(* CODESYS project WagoLibAwsIotThingShadow_v0.0.1.library
   Company: WAGO Corp. USA
   Title: WagoLibAwsIotThingShadow
   Description: This library contains function blocks which allow the project to interact directly with AWS IoT Thing Shadow document.
   Author: Jesse Cox
   Version: 0.0.1

Project tree, tasks and I/O mapping:
  libraries: SysProcess, 3.5.7.0 (System); WagoSysString, 1.6.0.0 (WAGO); WagoAppFileDir, * (WAGO); SysTypes2 Interfaces, 3.5.4.0 (System)
  text list GlobalTextList
  data type typIOT_THING_SHADOW
  function block GET_AWS_IOT_THING_SHADOW [ST]: CURL_STRING
  function block UPDATE_AWS_IOT_THING_SHADOW [ST]: PUB_STRING
*)

// typIOT_THING_SHADOW
TYPE typIOT_THING_SHADOW :
STRUCT
		sLabel	: STRING;
		sValue	: STRING;
END_STRUCT
END_TYPE

// GET_AWS_IOT_THING_SHADOW
FUNCTION_BLOCK GET_AWS_IOT_THING_SHADOW	
VAR_IN_OUT
	xExecute: BOOL;
	Shadow_Attributes	: ARRAY[*] OF typIOT_THING_SHADOW;
END_VAR
VAR_INPUT
	sThingName			: STRING;
	sRootCaPath			: STRING;
	sCertPath			: STRING;
	sKeyPath			: STRING;
	sEndpoint			: STRING;
END_VAR
VAR_OUTPUT
	//diTest				: DINT;
END_VAR
VAR
	sQueryBashScript	: STRING(255);
	sBashResponse: STRING;
	ptBashRslt: RTS_IEC_RESULT;
	diFileStatus: DINT;
	fbReadShadowFile: FbReadWholeFile_cpt;
	oReadFileStatus: FbResult;
	xReadFileTrig: BOOL;
	xREadFileError: BOOL;
	xREadFileBusy: BOOL;
	abFileData		: ARRAY[1..10000] OF BYTE;
	udiReadFileSize: UDINT := 10000;
	udiReadRxNumOfBytes: UDINT;
	xReadFileEndReached: BOOL;
	xConvertToTyp: BOOL;
	b: UDINT;
	xByteIsChar: BOOL;
	iCurlIndex: INT;
	xOnLabel: BOOL;
	xOnValue: BOOL;
	iWriteIndex: INT;
	sCurrentValueString: STRING;
	sCurrentLabelString: STRING;
	ub: DINT;
END_VAR

ub:=UPPER_BOUND (Shadow_Attributes,1);

IF xExecute THEN
	sQueryBashScript := CURL_STRING(
							sThingName:= sThingName, 
							sRootCaPath:= sRootCaPath, 
							sCertPath:= sCertPath, 
							sKeyPath:= sKeyPath, 
							sEndPoint:= sEndpoint);
	diFileStatus := SysProcessExecuteCommand2(pszCommand:= sQueryBashScript, pszStdOut:= sBashResponse, udiStdOutLen:= 255, pResult:= ptBashRslt);
	
	//diTest := diFileStatus;
	IF (diFileStatus <> 0) AND NOT xReadFileEndReached THEN
		xReadFileTrig := TRUE;
		fbReadShadowFile(
			oStatus=> oReadFileStatus, 
			xTrigger:= xReadFileTrig, 
			xError=> xREadFileError, 
			xBusy=> xREadFileBusy, 
			sName:= '/root/.rcv_shadow.json', 
			pRxBuffer:= ADR(abFileData), 
			udiRxBufferSize:= udiReadFileSize, 
			udiRxNBytes=> udiReadRxNumOfBytes, 
			xEofReached=> xReadFileEndReached);
			
			FOR b := 1 TO udiReadRxNumOfBytes DO
				//checks to see if the byte is an alpha-numeric
				IF 	((abFileData[b] >= 48) AND abFileData[b] <= 57) 	OR
					((abFileData[b] >= 65) AND abFileData[b] <= 90) 	OR
					((abFileData[b] >= 97) AND abFileData[b] <= 122) 	THEN
					xByteIsChar := TRUE;
				ELSE
					xByteIsChar := FALSE;
				END_IF
				
				// curly braces
				IF (abFileData[b] = 123) THEN
					iCurlIndex := iCurlIndex + 1;
				END_IF
				
				// if this is a new scan or the byte is a comma
				IF ((iCurlIndex = 3) AND (abFileData[b] = 123))  OR (abFileData[b] = 44) AND NOT xOnLabel THEN
					xOnLabel := TRUE;
					xOnValue := FALSE;
					Shadow_Attributes[iWriteIndex].sLabel:= sCurrentLabelString;
					Shadow_Attributes[iWriteIndex].sValue:= sCurrentValueString;
					sCurrentLabelString := '';
					sCurrentValueString := '';
					iWriteIndex := iWriteIndex + 1;
					
				//looks for a colon
				ELSIF (abFileData[b] = 58) THEN
					xOnLabel := FALSE;
					xOnValue := TRUE;
				END_IF
				
				IF xByteIsChar THEN
					IF xOnLabel THEN
						sCurrentLabelString := CONCAT(sCurrentLabelString, ASCIIBYTE_TO_STRING(abFileData[b]));
					ELSIF xOnValue THEN
						sCurrentValueString := CONCAT(sCurrentValueString, ASCIIBYTE_TO_STRING(abFileData[b]));
					END_IF
				END_IF

				IF iWriteIndex > ub THEN		
					// reseting variabel values here
					xReadFileEndReached := FALSE;
					xREadFileBusy := FALSE;
					xReadFileTrig := FALSE;
					xOnLabel := FALSE;
					xOnValue := FALSE;
					iCurlIndex := 0;
					iWriteIndex := 0;
					xExecute := FALSE;
				END_IF
			END_FOR
		END_IF
	//xExecute := FALSE;
END_IF

METHOD INTERNAL CURL_STRING : STRING(255)
VAR_INPUT
	sThingName	: STRING;
	sRootCaPath	: STRING;
	sCertPath	: STRING;
	sKeyPath	: STRING;
	sEndPoint	: STRING;
END_VAR

VAR
	sHoldString: STRING(255);
END_VAR
//sh .rcv_shadow.sh <root CA path> <certificate path> <private key path>  <endpoint>:8443/things/<thing name>/shadow
sHoldString := 'sh /root/.rcv_shadow.sh ';
sHoldString := CONCAT(sHoldString, sRootCaPath);
sHoldString := CONCAT(sHoldString, ' ');
sHoldString := CONCAT(sHoldString, sCertPath);
sHoldString := CONCAT(sHoldString, ' ');
sHoldString := CONCAT(sHoldString, sKeyPath);
sHoldString := CONCAT(sHoldString, ' ');
sHoldString := CONCAT(sHoldString, sEndpoint);
sHoldString := CONCAT(sHoldString, ':8443/things/');
sHoldString := CONCAT(sHoldString, sThingName);
sHoldString := CONCAT(sHoldString, '/shadow');

CURL_STRING := sHoldString;
END_METHOD

END_FUNCTION_BLOCK

// UPDATE_AWS_IOT_THING_SHADOW
FUNCTION_BLOCK UPDATE_AWS_IOT_THING_SHADOW
VAR_IN_OUT
	xExecute: BOOL;	// trigger to send the data to the AWS IoT Thing Shadow
	Shadow_Attributes	: ARRAY[*] OF typIOT_THING_SHADOW;
END_VAR
VAR_INPUT
	sRootCaPath			: STRING;
	sCertPath			: STRING;
	sKeyPath			: STRING;
	sEndpoint			: STRING;
	sTopic				: STRING;
END_VAR
VAR
	fbWriteFile			: FbWriteWholeFile_cpt;
	ub					: DINT;
	lb					: DINT;
	i					: DINT;
	sBaseString			: STRING(22) := '{"state":{"reported":{ ';
	sAttributeString	: STRING;
	aWriteBytes			: ARRAY[1..10000] OF BYTE;
	aHoldBytes			: ARRAY[1..80] OF BYTE;
	ptString 			: POINTER TO BYTE;
	l					: INT;
	diSizeOfString		: DINT;
	index				: INT;
	x: INT;
	sTestString: STRING(255);
	xWriteFile: BOOL;
	oWriteFileStatus: FbResult;
	xWriteFileTrig: BOOL;
	xWriteFileError: BOOL;
	xWriteFileBusy: BOOL;
	sWriteFileName: STRING := '/root/.send_shadow.json';
	sPublishBashScript: STRING(255);
	rtsSendResult: RTS_IEC_RESULT;
	sReturnResponse: STRING(255);
END_VAR

ub:=UPPER_BOUND (Shadow_Attributes,1);
lb:=LOWER_BOUND (Shadow_Attributes,1);

IF xExecute THEN
	index := 0;
	//begin building the array
	ptString := ADR(sBaseString);
	FOR l := 1 TO len(sBaseString) DO
		aWriteBytes[l] := ptString^;
		ptString := ptString + 1;
	END_FOR	
	ptString := 0;
	index := index + len(sBaseString);
	// write JSON header
	FOR i := lb TO ub DO /// loop through each atrribute / value
		sAttributeString := '"';
		sAttributeString := CONCAT(sAttributeString, Shadow_Attributes[i].sLabel);
		sAttributeString := CONCAT(sAttributeString, '": "');
		sAttributeString := CONCAT(sAttributeString, Shadow_Attributes[i].sValue);
		sAttributeString := CONCAT(sAttributeString, '"');
		IF (i < ub) THEN
			sAttributeString := CONCAT(sAttributeString, ',');
		ELSIF i = ub THEN
			sAttributeString := CONCAT(sAttributeString, '}}}');
		END_IF
		diSizeOfString := LEN(sAttributeString);
		ptString := ADR(sAttributeString);
		FOR l := 1 TO len(sAttributeString) DO
			aHoldBytes[l] := ptString^;
			ptString := ptString + 1;
			aWriteBytes[l + index] := aHoldBytes[l]; 
		END_FOR
		
		index := index + len(sAttributeString);
		
		IF i = ub THEN
			xWriteFileTrig := TRUE;
		END_IF
	END_FOR

// write the file
	fbWriteFile(
		oStatus=> oWriteFileStatus, 
		xTrigger:= xWriteFileTrig, 
		xError=> xWriteFileError, 
		xBusy=> xWriteFileBusy, 
		sName:= sWriteFileName, 
		pTxBuffer:= ADR(aWriteBytes), 
		udiTxNBytes:= index);
		
		IF NOT xWriteFileTrig THEN
			sPublishBashScript := PUB_STRING(
										sRootCaPath:= sRootCaPath, 
										sCertPath:= sCertPath, 
										sKeyPath:= sKeyPath, 
										sEndPoint:= sEndpoint, 
										sTopic:= sTopic);
			SysProcessExecuteCommand2(pszCommand:= sPublishBashScript, pszStdOut:= sReturnResponse, udiStdOutLen:= 255, pResult:= rtsSendResult);
			xExecute := FALSE;
		END_IF
END_IF

METHOD INTERNAL PUB_STRING : STRING(255)
VAR_INPUT
	sRootCaPath	: STRING;
	sCertPath	: STRING;
	sKeyPath	: STRING;
	sEndPoint	: STRING;
	sTopic		: STRING;
END_VAR

VAR
	sHoldString: STRING(255);
END_VAR
//mosquitto_pub --cafile (root ca cert)$1 --cert (certificate)$2 --key (private key)$3 -h (host address)$4 -p (port)8883 -q (qos)1 -d -t (topic)$5 -f (file to send)$6
sHoldString := 'sh /root/.send_shadow.sh ';
sHoldString := CONCAT(sHoldString, sRootCaPath);
sHoldString := CONCAT(sHoldString, ' ');
sHoldString := CONCAT(sHoldString, sCertPath);
sHoldString := CONCAT(sHoldString, ' ');
sHoldString := CONCAT(sHoldString, sKeyPath);
sHoldString := CONCAT(sHoldString, ' ');
sHoldString := CONCAT(sHoldString, sEndPoint);
sHoldString := CONCAT(sHoldString, ' $'');
sHoldString := CONCAT(sHoldString, sTopic);
sHoldString := CONCAT(sHoldString, '$' /root/.send_shadow.json');

PUB_STRING := sHoldString;
END_METHOD

END_FUNCTION_BLOCK
